FUNCTION_BLOCK AC
VAR_INPUT
END_VAR
VAR_OUTPUT
END_VAR
VAR
END_VAR

END_FUNCTION_BLOCK

(* stored: Version 1.1.0.1, ProductVersion 3.1.4024.13
   POU AC: Id {c4d831b3-90e1-4d32-9c0d-cbb508ea5eae}, SpecialFunc None *)
